Yaskawa INFORM job: LIGHT.JBI

/JOB
//NAME LIGHT
//POS
///NPOS 0,0,0,0,0,0
//INST
///DATE 2022/08/29 10:29
///ATTR SC,RW
///GROUP1 RB1
NOP
DOUT OT#(23) OFF
END
